PROGRAM MAIN
VAR
	res1Error: BOOL;
	Step: INT;
	Axis1_MV: MC_MoveVelocity;
	Axis1_Error_Reset: MC_Reset;
	Power1_BufferMode: MC_BufferMode;
	Power1_Override: LREAL;
	Power1_EnableNeg: BOOL;
	Power1_EnablePos: BOOL;
	Power1_Enable: BOOL;
	Axis1_Power: MC_Power;
	Axis1: AXIS_REF;
	Power1_Status: BOOL;
	Power1_Busy: BOOL;
	Power1_error: BOOL;
	Power1_Active: BOOL;
	Power1_ErrorID: UDINT;
	ErrorReset1_Execute: BOOL;
	res1Done: BOOL;
	res1Busy: BOOL;
	res1ErrorID: UDINT;
	MV1_Execute: BOOL;
	MV1_Done: BOOL;
	MV1_Velocity: LREAL;
	MV1_Decceleration: LREAL;
	MV1_Jerk: LREAL;
	MV1_Direction: MC_Direction;
	MV1_Buffermode: MC_BufferMode;
	MV1_InVelocity: BOOL;
	MV1_Busy: BOOL;
	MV1_CommandAborted: BOOL;
	MV1_Error: BOOL;
	MV1_ErrorID: UDINT;
	MV1_Acceleration: LREAL;
	MV1_Accelleration: LREAL;
	MV1_Active: BOOL;
	TorqueVAL AT %Q*: INT;
	TVAL  : INT;
	TorqueLim AT %Q*: UINT;
	Start1Btn: BOOL;
	PowerOnTorqueBtn: BOOL;
	Stop1Btn: BOOL;
	Setep: INT;
	TorqueEnable: BOOL;
	Axis2_Power: MC_Power;
	Axis2: AXIS_REF;
	Power2_EnablePos: BOOL;
	Power2_EnableNeg: BOOL;
	Power2_Enable: BOOL;
	Power2_Override: LREAL;
	Power2_BufferMode: MC_BufferMode;
	Power2_Status: BOOL;
	Power2_Busy: BOOL;
	Power2_Active: BOOL;
	Power2_Error: BOOL;
	Power2_ErrorID: UDINT;
	Axis2_ErrorReset: MC_Reset;
	ErrorReset2_Execute: BOOL;
	res2Done: BOOL;
	res2Busy: BOOL;
	res2Error: BOOL;
	res2ErrorID: UDINT;
	Axis2_MoveVelocity: MC_MoveVelocity;
	MV2_Execute: BOOL;
	MV2_Velocity: LREAL;
	MV2_Accelleration: LREAL;
	MV2_Decceleration: LREAL;
	MV2_Jerk: LREAL;
	MV2_Direction: MC_Direction;
	MV2_Buffermode: MC_BufferMode;
	MV2_InVelocity: BOOL;
	MV2_Busy: BOOL;
	MV2_Active: BOOL;
	MV2_CommandAborted: BOOL;
	MV2_Error: BOOL;
	MV2_ErrorID: UDINT;
	StepV: INT;
	PowerOnVelocityBtn: BOOL;
	Start2Btn: BOOL;
	Stop2Btn: BOOL;
	MVelocity: INT;
END_VAR

//Axis1 - Torque controlled servomotor
//Axis2 - Velocity controlled servomotor
Axis1_Power(
	Axis:=Axis1,
	Enable := Power1_Enable,
	Enable_Positive := Power1_EnablePos,
	Enable_Negative := Power1_EnableNeg,
	Override := Power1_Override,
	BufferMode := Power1_BufferMode,
	Status => Power1_Status,
	Busy => Power1_Busy,
	Active => Power1_Active,
	Error => Power1_error,
	ErrorID =>Power1_ErrorID);
	
Axis2_Power(
	Axis:= Axis2, 
	Enable:= Power2_Enable, 
	Enable_Positive:= Power2_EnablePos, 
	Enable_Negative:= Power2_EnableNeg, 
	Override:= Power2_Override, 
	BufferMode:= Power2_BufferMode, 
	//Options:= , 
	Status=> Power2_Status, 
	Busy=> Power2_Busy, 
	Active=> Power2_Active, 
	Error=> Power2_Error, 
	ErrorID=> Power2_ErrorID);
	
Axis1_Error_Reset(
	Axis := Axis1,
	Execute := ErrorReset1_Execute,
	Done => res1Done,
	Busy => res1Busy,
	Error => res1Error,
	ErrorID => res1ErrorID);
	
Axis2_ErrorReset(
	Axis := Axis2,
	Execute := ErrorReset2_Execute,
	Done => res2Done,
	Busy => res2Busy,
	Error => res2Error,
	ErrorID => res2ErrorID);
	
Axis1_MV(
	Axis:= Axis1, 
	Execute:= MV1_Execute, 
	Velocity:= MV1_Velocity, 
	Acceleration:= MV1_Accelleration, 
	Deceleration:= MV1_Decceleration, 
	Jerk:= MV1_Jerk, 
	Direction:= MV1_Direction, 
	BufferMode:= MV1_Buffermode, 
	//Options:= MV_Options, 
	InVelocity=> MV1_InVelocity, 
	Busy=> MV1_Busy, 
	Active=> MV1_Active, 
	CommandAborted=> MV1_CommandAborted, 
	Error=> MV1_Error, 
	ErrorID=> MV1_ErrorID);
	
Axis2_MoveVelocity(
	Axis:= Axis2, 
	Execute:= MV2_Execute, 
	Velocity:= MV2_Velocity, 
	Acceleration:= MV2_Accelleration, 
	Deceleration:= MV2_Decceleration, 
	Jerk:= MV2_Jerk, 
	Direction:= MV2_Direction, 
	BufferMode:= MV2_Buffermode, 
	//Options:= MV_Options, 
	InVelocity=> MV2_InVelocity, 
	Busy=> MV2_Busy, 
	Active=> MV2_Active, 
	CommandAborted=> MV2_CommandAborted, 
	Error=> MV2_Error, 
	ErrorID=> MV2_ErrorID);
	
	//Torque Controlled Servo
	
	//In case of an error with torque controlled servo:
	IF(Power1_error = TRUE OR MV1_Error=TRUE)THEN
		Step := 10;
	END_IF
	
	//Enables user to set the torque of the servomotor
	IF TorqueEnable  = TRUE THEN
		TorqueVAL := TVAL;
	END_IF
	CASE Step OF
		0://Start of the power (in next step), when the PowerOnTorque button will be clicked
			IF (PowerOnTorqueBtn = TRUE) THEN
				Setep := 1;
			END_IF
		1://Start the torque control, when the StartTorque button will be clicked
			Power1_Enable := TRUE;
			Power1_EnablePos := TRUE;
			Power1_EnableNeg := TRUE;
			Power1_Override := 100;
			PowerOnTorqueBtn := FALSE;
			IF (Start1Btn = TRUE) THEN
				Step := 2;
			END_IF
		2://Stop the motor (in next step), when the StopTorque button will be clicked
			MV1_Execute := TRUE; 
			MV1_Velocity := 100; 
			MV1_Accelleration := 100; 
			MV1_Decceleration := 100;
			MV1_Jerk := 100;
			TorqueLim := 1000;
			TorqueEnable := TRUE;
			Start1Btn := FALSE;
			IF Stop1Btn = TRUE THEN
				Step:= 3;
				
			END_IF
		3://Stops motor and gets back to the Power On state
			IF TorqueVAL = 0 THEN
				MV1_Execute := TRUE;
				Step := 1;
			END_IF
			MV1_Execute := FALSE;
			MV1_Velocity := 0;
			TorqueEnable := FALSE;
			TorqueVAL := 0;
			Stop1Btn := FALSE;
			
		10://Error Step
			Power1_Enable := FALSE;
			MV1_Execute := FALSE; 
			MV1_Velocity := 0;
			TorqueVAL := 0;
			TorqueEnable := FALSE;
			ErrorReset1_Execute := TRUE;
			IF res1Done = TRUE THEN
				Step := 0;
			END_IF
			
		END_CASE
		
		//Velocity Controlled Servo
		
		//In case of an error with torque controlled servo:
	IF(Power2_error = TRUE OR MV2_Error=TRUE) THEN
		StepV := 10;
	END_IF
		
		CASE StepV OF
		0://Start of the power (in next step), when the PowerOnVelocity button will be clicked
			IF (PowerOnVelocityBtn = TRUE) THEN
				StepV := 1;
			END_IF
		1://Start the torque control, when the StartTorque button will be clicked
			Power2_Enable := TRUE;
			Power2_EnablePos := TRUE;
			Power2_EnableNeg := TRUE;
			Power2_Override := 100;
			PowerOnVelocityBtn := FALSE;
			IF (Start2Btn = TRUE) THEN
				StepV := 2;
			END_IF
		2://Stop the motor (in next step), when the StopVelocity button will be clicked
			MV2_Execute := TRUE; 
			
			IF NOT(MV2_Velocity = MVelocity) THEN
				MV2_Velocity := MVelocity;
				MV2_Execute := FALSE; 
			END_IF
			 
			MV2_Accelleration := 100; 
			MV2_Decceleration := 100;
			MV2_Jerk := 100;
			Start2Btn := FALSE;
			IF Stop2Btn = TRUE THEN
				StepV:= 3;
			END_IF
		3://Stops motor and gets back to the Power On state
			IF MV2_Velocity = 0 THEN
				MV1_Execute := TRUE;
				StepV := 1;
			END_IF
			MV2_Execute := FALSE;
			MV2_Velocity := 0;
			Stop2Btn := FALSE;
						
			
		10://Error Step
			Power2_Enable := FALSE;
			MV2_Execute := FALSE; 
			MV2_Velocity := 0;
			ErrorReset2_Execute := TRUE;
			IF res2Done = TRUE THEN
				StepV := 0;
			END_IF
			
		END_CASE

END_PROGRAM

(* stored: Version 1.1.0.1, ProductVersion 3.1.4024.4
   POU MAIN: Id {1da18359-142c-4771-bf7e-d261e8caea2a}, SpecialFunc None *)
